TYPE "PTrk_Item"
VERSION : 0.1
// Block: PTrk_Item
   STRUCT
      P_ID : DInt;
      O_ID : DInt;
      C_ID : DInt;
      Quality : Int;
      Beam_Code : Int;
      PLen_Meas : Real;
      W_A : Real;
      H_B : Real;
      ShiftDone : Bool;
   END_STRUCT;

END_TYPE
